SUBAPPLICATION Uebung_001c3 (* DigitalInput_I1 auf DigitalOutput_Q1 --> Eingang abfragen bei Boot. *)
  (* Standard: 61499-2; Description: Copyright (c) 2023 Meisterschulen am Ostbahnhof This program and the accompanying materials are made available under the terms of the Eclipse Public License 2.0 which is available at https://www.eclipse.org/legal/epl-2.0/ SPDX-License-Identifier: EPL-2.0 *)
  (* Version 1.0, 2023-10-23, Franz Höpfinger, Meisterschulen am Ostbahnhof, initial API and implementation and/or initial documentation *)
  PACKAGE Uebungen;
  IMPORT logiBUS::io::DI::logiBUS_DI::Input_I1;
  IMPORT logiBUS::io::DQ::logiBUS_DO::Output_Q1;
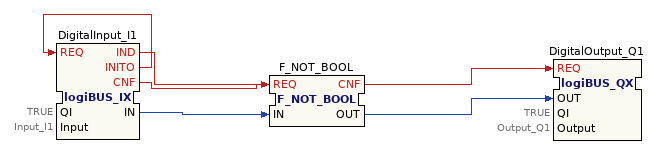
  (* ohne die Linie INITO->REQ ist der Ausgang Q1 beim Start FALSE. mit der Linie ist er TRUE. *)
  (* "Negate Connection" mach ein NOT am Eingang; das geht nur bei BOOL. --> hier wird aus dem F_NOT_BOOL dann ein NOOP. *)
  FBS
    DigitalOutput_Q1 : logiBUS::io::DQ::logiBUS_QX(QI := TRUE, Output := Output_Q1);
    DigitalInput_I1 : logiBUS::io::DI::logiBUS_IX(QI := TRUE, Input := Input_I1);
    F_NOT_BOOL : iec61131::booleanOperators::F_NOT_BOOL;
  END_FBS
  EVENT_CONNECTIONS
    DigitalInput_I1.IND TO F_NOT_BOOL.REQ;
    DigitalInput_I1.INITO TO DigitalInput_I1.REQ;
    DigitalInput_I1.CNF TO F_NOT_BOOL.REQ;
    F_NOT_BOOL.CNF TO DigitalOutput_Q1.REQ;
  END_CONNECTIONS
  DATA_CONNECTIONS
    DigitalInput_I1.IN TO F_NOT_BOOL.IN; {SET_ATTRIBUTE(Negated, true)}
    F_NOT_BOOL.OUT TO DigitalOutput_Q1.OUT;
  END_CONNECTIONS
END_SUBAPPLICATION
